// TIA Portal V16 export
// export: Created 2022-11-17T11:55:01.3238925Z, ExportSetting WithDefaults, DisplayName Totally Integrated Automation Portal, DisplayVersion V16 Update 6, DisplayName TIA Portal Version Control Interface, DisplayVersion V16 Update 2, DisplayName TIA Portal Openness, DisplayVersion V16 Update 6, DisplayName SINAMICS Startdrive Advanced, DisplayVersion V16 Update 5, DisplayName SINAMICS Startdrive G130, G150, S120, S150, SINAMICS MV, S210, DisplayVersion V16 Update 5, DisplayName SINAMICS Startdrive G110M, G120, G120C, G120D, G120P, G115D, DisplayVersion V16 Update 5, DisplayName STEP 7 Professional, DisplayVersion V16 Update 6, DisplayName STEP 7 Safety, DisplayVersion V16, DisplayName WinCC Advanced, DisplayVersion V16 Update 6
FUNCTION "FC01_SupportOut" : Void   // FC1, LAD
TITLE = Output support memory
{ S7_Optimized_Access := 'FALSE' }
AUTHOR : Robopac
VERSION : 0.0
// stored: AutoNumber false, IsIECCheckEnabled false, SetENOAutomatically false, UDAEnableTagReadback false
BEGIN

REGION Network 1: STANDARD
END_REGION

REGION Network 2: Emergency mode lamp (Technoplat)
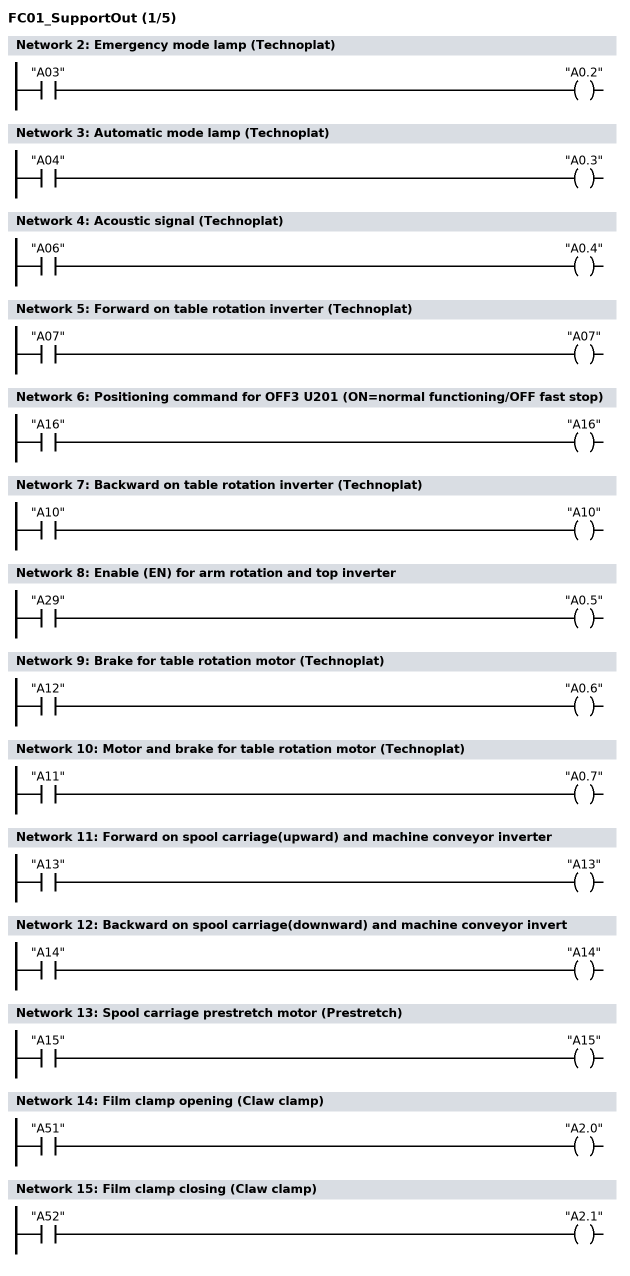
   RUNG wire#powerrail
      Contact( "A03" )
      Coil( "A0.2" )
   END_RUNG
   // the same network as SCL:
   "A0.2" := "A03";
END_REGION

REGION Network 3: Automatic mode lamp (Technoplat)
   RUNG wire#powerrail
      Contact( "A04" )
      Coil( "A0.3" )
   END_RUNG
   // the same network as SCL:
   "A0.3" := "A04";
END_REGION

REGION Network 4: Acoustic signal (Technoplat)
   RUNG wire#powerrail
      Contact( "A06" )
      Coil( "A0.4" )
   END_RUNG
   // the same network as SCL:
   "A0.4" := "A06";
END_REGION

REGION Network 5: Forward on table rotation inverter (Technoplat)
   RUNG wire#powerrail
      Contact( "A07" )
      Coil( "A07" )
   END_RUNG
   // the same network as SCL:
   "A07" := "A07";
END_REGION

REGION Network 6: Positioning command for OFF3 U201 (ON=normal functioning/OFF fast stop)
   RUNG wire#powerrail
      Contact( "A16" )
      Coil( "A16" )
   END_RUNG
   // the same network as SCL:
   "A16" := "A16";
END_REGION

REGION Network 7: Backward on table rotation inverter (Technoplat)
   RUNG wire#powerrail
      Contact( "A10" )
      Coil( "A10" )
   END_RUNG
   // the same network as SCL:
   "A10" := "A10";
END_REGION

REGION Network 8: Enable (EN) for arm rotation and top inverter
   RUNG wire#powerrail
      Contact( "A29" )
      Coil( "A0.5" )
   END_RUNG
   // the same network as SCL:
   "A0.5" := "A29";
END_REGION

REGION Network 9: Brake for table rotation motor (Technoplat)
   RUNG wire#powerrail
      Contact( "A12" )
      Coil( "A0.6" )
   END_RUNG
   // the same network as SCL:
   "A0.6" := "A12";
END_REGION

REGION Network 10: Motor and brake for table rotation motor (Technoplat)
   RUNG wire#powerrail
      Contact( "A11" )
      Coil( "A0.7" )
   END_RUNG
   // the same network as SCL:
   "A0.7" := "A11";
END_REGION

REGION Network 11: Forward on spool carriage(upward) and machine conveyor inverter
   RUNG wire#powerrail
      Contact( "A13" )
      Coil( "A13" )
   END_RUNG
   // the same network as SCL:
   "A13" := "A13";
END_REGION

REGION Network 12: Backward on spool carriage(downward) and machine conveyor invert
   RUNG wire#powerrail
      Contact( "A14" )
      Coil( "A14" )
   END_RUNG
   // the same network as SCL:
   "A14" := "A14";
END_REGION

REGION Network 13: Spool carriage prestretch motor (Prestretch)
   RUNG wire#powerrail
      Contact( "A15" )
      Coil( "A15" )
   END_RUNG
   // the same network as SCL:
   "A15" := "A15";
END_REGION

REGION Network 14: Film clamp opening (Claw clamp)
   RUNG wire#powerrail
      Contact( "A51" )
      Coil( "A2.0" )
   END_RUNG
   // the same network as SCL:
   "A2.0" := "A51";
END_REGION

REGION Network 15: Film clamp closing (Claw clamp)
   RUNG wire#powerrail
      Contact( "A52" )
      Coil( "A2.1" )
   END_RUNG
   // the same network as SCL:
   "A2.1" := "A52";
END_REGION

REGION Network 16: Cutting and welding unit forward(1)/backward (Claw clamp)
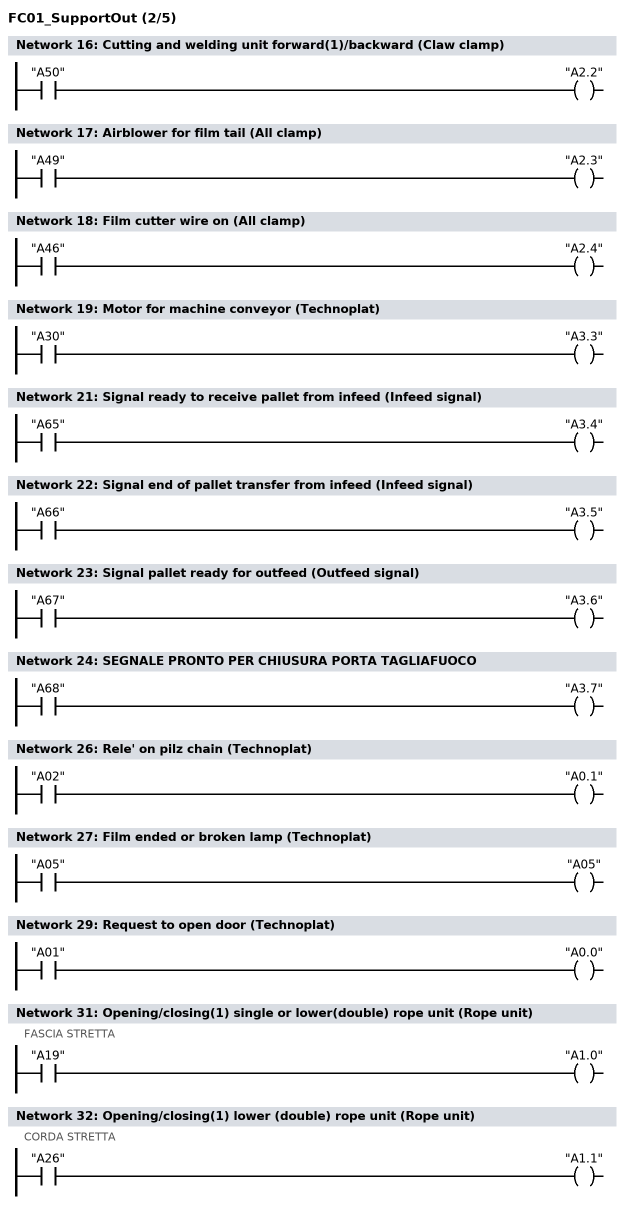
   RUNG wire#powerrail
      Contact( "A50" )
      Coil( "A2.2" )
   END_RUNG
   // the same network as SCL:
   "A2.2" := "A50";
END_REGION

REGION Network 17: Airblower for film tail (All clamp)
   RUNG wire#powerrail
      Contact( "A49" )
      Coil( "A2.3" )
   END_RUNG
   // the same network as SCL:
   "A2.3" := "A49";
END_REGION

REGION Network 18: Film cutter wire on (All clamp)
   RUNG wire#powerrail
      Contact( "A46" )
      Coil( "A2.4" )
   END_RUNG
   // the same network as SCL:
   "A2.4" := "A46";
END_REGION

REGION Network 19: Motor for machine conveyor (Technoplat)
   RUNG wire#powerrail
      Contact( "A30" )
      Coil( "A3.3" )
   END_RUNG
   // the same network as SCL:
   "A3.3" := "A30";
END_REGION

REGION Network 20: EXCHANGE SIGNALS
END_REGION

REGION Network 21: Signal ready to receive pallet from infeed (Infeed signal)
   RUNG wire#powerrail
      Contact( "A65" )
      Coil( "A3.4" )
   END_RUNG
   // the same network as SCL:
   "A3.4" := "A65";
END_REGION

REGION Network 22: Signal end of pallet transfer from infeed (Infeed signal)
   RUNG wire#powerrail
      Contact( "A66" )
      Coil( "A3.5" )
   END_RUNG
   // the same network as SCL:
   "A3.5" := "A66";
END_REGION

REGION Network 23: Signal pallet ready for outfeed (Outfeed signal)
   RUNG wire#powerrail
      Contact( "A67" )
      Coil( "A3.6" )
   END_RUNG
   // the same network as SCL:
   "A3.6" := "A67";
END_REGION

REGION Network 24: SEGNALE PRONTO PER CHIUSURA PORTA TAGLIAFUOCO
   RUNG wire#powerrail
      Contact( "A68" )
      Coil( "A3.7" )
   END_RUNG
   // the same network as SCL:
   "A3.7" := "A68";
END_REGION

REGION Network 25: ACCESSORIES
END_REGION

REGION Network 26: Rele' on pilz chain (Technoplat)
   RUNG wire#powerrail
      Contact( "A02" )
      Coil( "A0.1" )
   END_RUNG
   // the same network as SCL:
   "A0.1" := "A02";
END_REGION

REGION Network 27: Film ended or broken lamp (Technoplat)
   RUNG wire#powerrail
      Contact( "A05" )
      Coil( "A05" )
   END_RUNG
   // the same network as SCL:
   "A05" := "A05";
END_REGION

REGION Network 28: ***DOOR***
END_REGION

REGION Network 29: Request to open door (Technoplat)
   RUNG wire#powerrail
      Contact( "A01" )
      Coil( "A0.0" )
   END_RUNG
   // the same network as SCL:
   "A0.0" := "A01";
END_REGION

REGION Network 30: ***BAND/ROPE***
END_REGION

REGION Network 31: Opening/closing(1) single or lower(double) rope unit (Rope unit)
   // FASCIA STRETTA
   RUNG wire#powerrail
      Contact( "A19" )
      Coil( "A1.0" )
   END_RUNG
   // the same network as SCL:
   "A1.0" := "A19";
END_REGION

REGION Network 32: Opening/closing(1) lower (double) rope unit (Rope unit)
   // CORDA STRETTA
   RUNG wire#powerrail
      Contact( "A26" )
      Coil( "A1.1" )
   END_RUNG
   // the same network as SCL:
   "A1.1" := "A26";
END_REGION

REGION Network 33: ***WELDER***
END_REGION

REGION Network 34: Film welder on (All clamp)
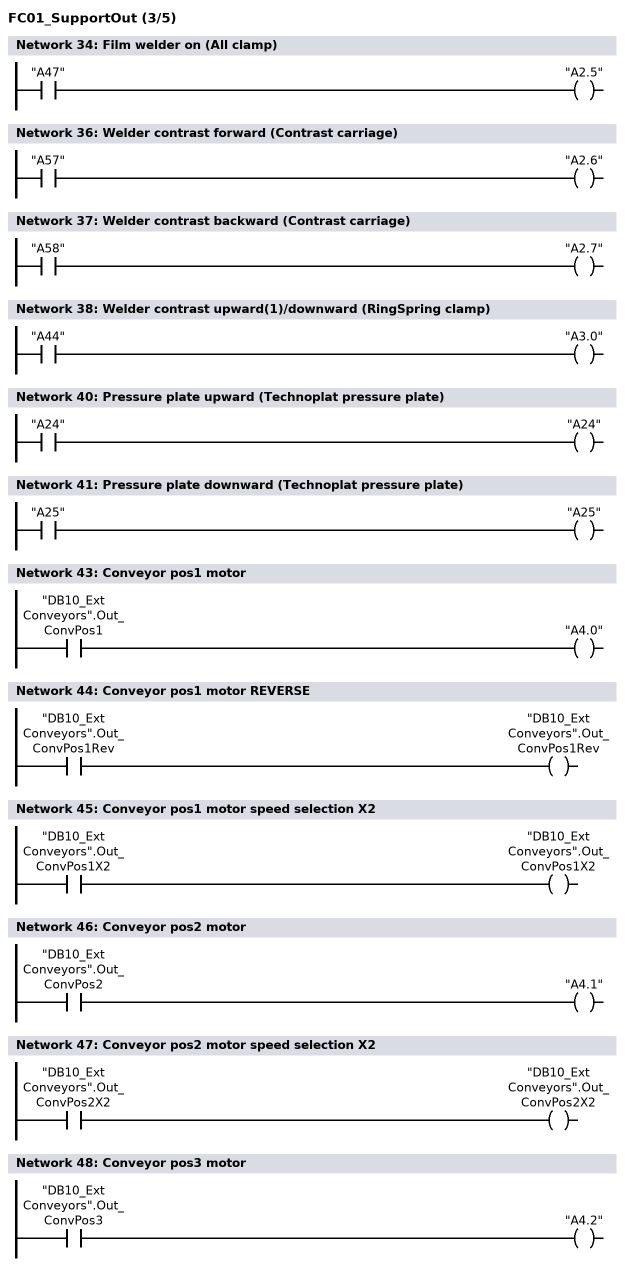
   RUNG wire#powerrail
      Contact( "A47" )
      Coil( "A2.5" )
   END_RUNG
   // the same network as SCL:
   "A2.5" := "A47";
END_REGION

REGION Network 35: ***CONTRAST***
END_REGION

REGION Network 36: Welder contrast forward (Contrast carriage)
   RUNG wire#powerrail
      Contact( "A57" )
      Coil( "A2.6" )
   END_RUNG
   // the same network as SCL:
   "A2.6" := "A57";
END_REGION

REGION Network 37: Welder contrast backward (Contrast carriage)
   RUNG wire#powerrail
      Contact( "A58" )
      Coil( "A2.7" )
   END_RUNG
   // the same network as SCL:
   "A2.7" := "A58";
END_REGION

REGION Network 38: Welder contrast upward(1)/downward (RingSpring clamp)
   RUNG wire#powerrail
      Contact( "A44" )
      Coil( "A3.0" )
   END_RUNG
   // the same network as SCL:
   "A3.0" := "A44";
END_REGION

REGION Network 39: ***PRESSURE***
END_REGION

REGION Network 40: Pressure plate upward (Technoplat pressure plate)
   RUNG wire#powerrail
      Contact( "A24" )
      Coil( "A24" )
   END_RUNG
   // the same network as SCL:
   "A24" := "A24";
END_REGION

REGION Network 41: Pressure plate downward (Technoplat pressure plate)
   RUNG wire#powerrail
      Contact( "A25" )
      Coil( "A25" )
   END_RUNG
   // the same network as SCL:
   "A25" := "A25";
END_REGION

REGION Network 42: ***CONVEYORS***
END_REGION

REGION Network 43: Conveyor pos1 motor
   RUNG wire#powerrail
      Contact( "DB10_ExtConveyors".Out_ConvPos1 )
      Coil( "A4.0" )
   END_RUNG
   // the same network as SCL:
   "A4.0" := "DB10_ExtConveyors".Out_ConvPos1;
END_REGION

REGION Network 44: Conveyor pos1 motor REVERSE
   RUNG wire#powerrail
      Contact( "DB10_ExtConveyors".Out_ConvPos1Rev )
      Coil( "DB10_ExtConveyors".Out_ConvPos1Rev )
   END_RUNG
   // the same network as SCL:
   "DB10_ExtConveyors".Out_ConvPos1Rev := "DB10_ExtConveyors".Out_ConvPos1Rev;
END_REGION

REGION Network 45: Conveyor pos1 motor speed selection X2
   RUNG wire#powerrail
      Contact( "DB10_ExtConveyors".Out_ConvPos1X2 )
      Coil( "DB10_ExtConveyors".Out_ConvPos1X2 )
   END_RUNG
   // the same network as SCL:
   "DB10_ExtConveyors".Out_ConvPos1X2 := "DB10_ExtConveyors".Out_ConvPos1X2;
END_REGION

REGION Network 46: Conveyor pos2 motor
   RUNG wire#powerrail
      Contact( "DB10_ExtConveyors".Out_ConvPos2 )
      Coil( "A4.1" )
   END_RUNG
   // the same network as SCL:
   "A4.1" := "DB10_ExtConveyors".Out_ConvPos2;
END_REGION

REGION Network 47: Conveyor pos2 motor speed selection X2
   RUNG wire#powerrail
      Contact( "DB10_ExtConveyors".Out_ConvPos2X2 )
      Coil( "DB10_ExtConveyors".Out_ConvPos2X2 )
   END_RUNG
   // the same network as SCL:
   "DB10_ExtConveyors".Out_ConvPos2X2 := "DB10_ExtConveyors".Out_ConvPos2X2;
END_REGION

REGION Network 48: Conveyor pos3 motor
   RUNG wire#powerrail
      Contact( "DB10_ExtConveyors".Out_ConvPos3 )
      Coil( "A4.2" )
   END_RUNG
   // the same network as SCL:
   "A4.2" := "DB10_ExtConveyors".Out_ConvPos3;
END_REGION

REGION Network 49: Conveyor pos4 motor
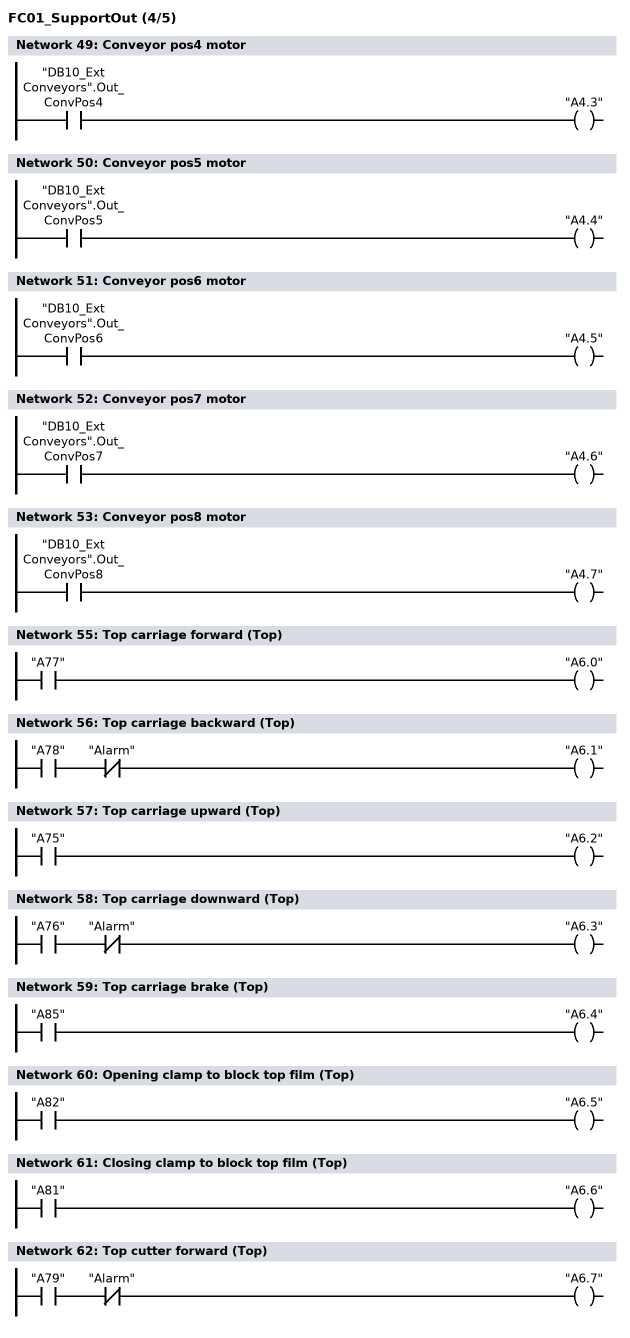
   RUNG wire#powerrail
      Contact( "DB10_ExtConveyors".Out_ConvPos4 )
      Coil( "A4.3" )
   END_RUNG
   // the same network as SCL:
   "A4.3" := "DB10_ExtConveyors".Out_ConvPos4;
END_REGION

REGION Network 50: Conveyor pos5 motor
   RUNG wire#powerrail
      Contact( "DB10_ExtConveyors".Out_ConvPos5 )
      Coil( "A4.4" )
   END_RUNG
   // the same network as SCL:
   "A4.4" := "DB10_ExtConveyors".Out_ConvPos5;
END_REGION

REGION Network 51: Conveyor pos6 motor
   RUNG wire#powerrail
      Contact( "DB10_ExtConveyors".Out_ConvPos6 )
      Coil( "A4.5" )
   END_RUNG
   // the same network as SCL:
   "A4.5" := "DB10_ExtConveyors".Out_ConvPos6;
END_REGION

REGION Network 52: Conveyor pos7 motor
   RUNG wire#powerrail
      Contact( "DB10_ExtConveyors".Out_ConvPos7 )
      Coil( "A4.6" )
   END_RUNG
   // the same network as SCL:
   "A4.6" := "DB10_ExtConveyors".Out_ConvPos7;
END_REGION

REGION Network 53: Conveyor pos8 motor
   RUNG wire#powerrail
      Contact( "DB10_ExtConveyors".Out_ConvPos8 )
      Coil( "A4.7" )
   END_RUNG
   // the same network as SCL:
   "A4.7" := "DB10_ExtConveyors".Out_ConvPos8;
END_REGION

REGION Network 54: ***TOP***
END_REGION

REGION Network 55: Top carriage forward (Top)
   RUNG wire#powerrail
      Contact( "A77" )
      Coil( "A6.0" )
   END_RUNG
   // the same network as SCL:
   "A6.0" := "A77";
END_REGION

REGION Network 56: Top carriage backward (Top)
   RUNG wire#powerrail
      Contact( "A78" )
      I_Contact( "Alarm" )
      Coil( "A6.1" )
   END_RUNG
   // the same network as SCL:
   "A6.1" := "A78" AND NOT "Alarm";
END_REGION

REGION Network 57: Top carriage upward (Top)
   RUNG wire#powerrail
      Contact( "A75" )
      Coil( "A6.2" )
   END_RUNG
   // the same network as SCL:
   "A6.2" := "A75";
END_REGION

REGION Network 58: Top carriage downward (Top)
   RUNG wire#powerrail
      Contact( "A76" )
      I_Contact( "Alarm" )
      Coil( "A6.3" )
   END_RUNG
   // the same network as SCL:
   "A6.3" := "A76" AND NOT "Alarm";
END_REGION

REGION Network 59: Top carriage brake (Top)
   RUNG wire#powerrail
      Contact( "A85" )
      Coil( "A6.4" )
   END_RUNG
   // the same network as SCL:
   "A6.4" := "A85";
END_REGION

REGION Network 60: Opening clamp to block top film (Top)
   RUNG wire#powerrail
      Contact( "A82" )
      Coil( "A6.5" )
   END_RUNG
   // the same network as SCL:
   "A6.5" := "A82";
END_REGION

REGION Network 61: Closing clamp to block top film (Top)
   RUNG wire#powerrail
      Contact( "A81" )
      Coil( "A6.6" )
   END_RUNG
   // the same network as SCL:
   "A6.6" := "A81";
END_REGION

REGION Network 62: Top cutter forward (Top)
   RUNG wire#powerrail
      Contact( "A79" )
      I_Contact( "Alarm" )
      Coil( "A6.7" )
   END_RUNG
   // the same network as SCL:
   "A6.7" := "A79" AND NOT "Alarm";
END_REGION

REGION Network 63: Top cutter backward (Top)
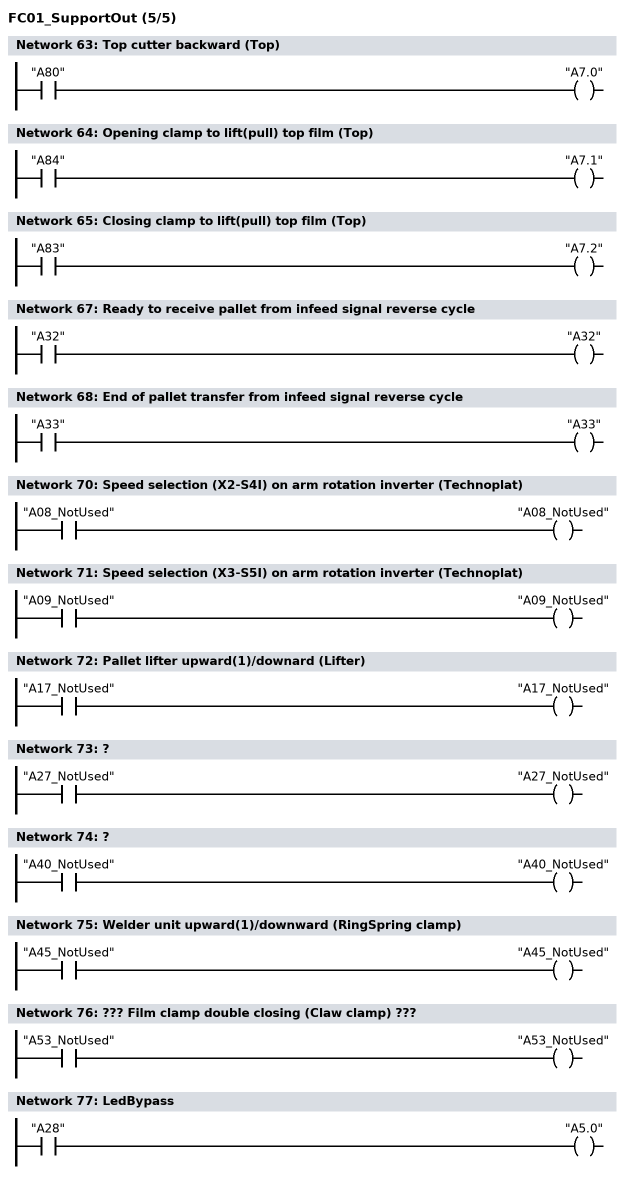
   RUNG wire#powerrail
      Contact( "A80" )
      Coil( "A7.0" )
   END_RUNG
   // the same network as SCL:
   "A7.0" := "A80";
END_REGION

REGION Network 64: Opening clamp to lift(pull) top film (Top)
   RUNG wire#powerrail
      Contact( "A84" )
      Coil( "A7.1" )
   END_RUNG
   // the same network as SCL:
   "A7.1" := "A84";
END_REGION

REGION Network 65: Closing clamp to lift(pull) top film (Top)
   RUNG wire#powerrail
      Contact( "A83" )
      Coil( "A7.2" )
   END_RUNG
   // the same network as SCL:
   "A7.2" := "A83";
END_REGION

REGION Network 66: OTHER
END_REGION

REGION Network 67: Ready to receive pallet from infeed signal reverse cycle
   RUNG wire#powerrail
      Contact( "A32" )
      Coil( "A32" )
   END_RUNG
   // the same network as SCL:
   "A32" := "A32";
END_REGION

REGION Network 68: End of pallet transfer from infeed signal reverse cycle
   RUNG wire#powerrail
      Contact( "A33" )
      Coil( "A33" )
   END_RUNG
   // the same network as SCL:
   "A33" := "A33";
END_REGION

REGION Network 69: OLD (NOT USED)
END_REGION

REGION Network 70: Speed selection (X2-S4I) on arm rotation inverter (Technoplat)
   RUNG wire#powerrail
      Contact( "A08_NotUsed" )
      Coil( "A08_NotUsed" )
   END_RUNG
   // the same network as SCL:
   "A08_NotUsed" := "A08_NotUsed";
END_REGION

REGION Network 71: Speed selection (X3-S5I) on arm rotation inverter (Technoplat)
   RUNG wire#powerrail
      Contact( "A09_NotUsed" )
      Coil( "A09_NotUsed" )
   END_RUNG
   // the same network as SCL:
   "A09_NotUsed" := "A09_NotUsed";
END_REGION

REGION Network 72: Pallet lifter upward(1)/downard (Lifter)
   RUNG wire#powerrail
      Contact( "A17_NotUsed" )
      Coil( "A17_NotUsed" )
   END_RUNG
   // the same network as SCL:
   "A17_NotUsed" := "A17_NotUsed";
END_REGION

REGION Network 73: ?
   RUNG wire#powerrail
      Contact( "A27_NotUsed" )
      Coil( "A27_NotUsed" )
   END_RUNG
   // the same network as SCL:
   "A27_NotUsed" := "A27_NotUsed";
END_REGION

REGION Network 74: ?
   RUNG wire#powerrail
      Contact( "A40_NotUsed" )
      Coil( "A40_NotUsed" )
   END_RUNG
   // the same network as SCL:
   "A40_NotUsed" := "A40_NotUsed";
END_REGION

REGION Network 75: Welder unit upward(1)/downward (RingSpring clamp)
   RUNG wire#powerrail
      Contact( "A45_NotUsed" )
      Coil( "A45_NotUsed" )
   END_RUNG
   // the same network as SCL:
   "A45_NotUsed" := "A45_NotUsed";
END_REGION

REGION Network 76: ??? Film clamp double closing (Claw clamp) ???
   RUNG wire#powerrail
      Contact( "A53_NotUsed" )
      Coil( "A53_NotUsed" )
   END_RUNG
   // the same network as SCL:
   "A53_NotUsed" := "A53_NotUsed";
END_REGION

REGION Network 77: LedBypass
   RUNG wire#powerrail
      Contact( "A28" )
      Coil( "A5.0" )
   END_RUNG
   // the same network as SCL:
   "A5.0" := "A28";
END_REGION
END_FUNCTION
